FUNCTION INTERNAL F_IsSystemValid : BOOL
VAR_STAT
	{attribute 'hide'}
	fbTcConfig		: TC_Config;	
	{attribute 'hide'}
	bIsRequested 	: BOOL;
	{attribute 'hide'}
	bIsSystemValid	: BOOL;
END_VAR

IF NOT bIsRequested THEN
	IF NOT __ISVALIDREF(GVL_Core.refSystem) THEN	
		ADSLOGSTR(msgCtrlMask := ADSLOG_MSGTYPE_ERROR OR ADSLOG_MSGTYPE_MSGBOX, 'OC: %s', 'FB_System can not be found! TwinCAT is switched to Config Mode');
		fbTcConfig(NETID := '', SET := TRUE);
		bIsSystemValid := FALSE;
	ELSE
		bIsSystemValid := TRUE;
	END_IF
END_IF

bIsRequested := TRUE;
F_IsSystemValid := bIsSystemValid;

END_FUNCTION

(* stored: Version 1.1.0.1, ProductVersion 3.1.4024.12
   POU F_IsSystemValid: Id {b0a17754-8ecf-0688-0d46-47efa9bc4fda}, SpecialFunc None *)
